# EPICS autosave request: filter/auto_settings.req
# Kohzu monochromator
#file kohzuSeq_settings.req P=$(P)

# High resolution monochromator
#file hrSeq_settings.req P=$(P),N=1

# Io calc
#file Io_settings.req P=xxx:Io:

# orientation matrix
#file orient_settings.req P=$(P),O=1
#file orient_xtals_settings.req P=$(P),O=1

### PID_based feedback
#file fb_epid.req P=$(P)epid1

#file SGM_settings.req P=$(P),SGM=SGM1

file filterDrive.req "P=BL172:,R=filter:"
file filterBladeNoSensor.req "P=BL172:,R=filter:,N=1"
file filterBladeNoSensor.req "P=BL172:,R=filter:,N=2"
file filterBladeNoSensor.req "P=BL172:,R=filter:,N=3"
file filterBladeNoSensor.req "P=BL172:,R=filter:,N=4"
